// TIA Portal V17 export
// export: Created 2022-07-20T07:01:31.3759363Z, ExportSetting WithDefaults, DisplayName Totally Integrated Automation Portal, DisplayVersion V17, DisplayName TIA Portal Openness, DisplayVersion V17, DisplayName TIA Portal Version Control Interface, DisplayVersion V17, DisplayName SINAMICS Startdrive Advanced, DisplayVersion V17, DisplayName SINAMICS Startdrive G130, G150, S120, S150, SINAMICS MV, S210, DisplayVersion V17, DisplayName SINAMICS Startdrive G110M, G120, G120C, G120D, G120P, G115D, DisplayVersion V17, DisplayName STEP 7 Professional, DisplayVersion V17, DisplayName STEP 7 Safety, DisplayVersion V17, DisplayName WinCC Advanced, DisplayVersion V17
FUNCTION "FC10330_2BytesToUDint" : UDInt   // FC10330, LAD
{ S7_Optimized_Access := 'TRUE' }
VERSION : 0.1
// stored: AutoNumber false, IsIECCheckEnabled false, SetENOAutomatically false, UDAEnableTagReadback false
   VAR_INPUT
      LowByte : Byte;
      HighByte : Byte;
   END_VAR
BEGIN

REGION Network 1 (SCL): 2 Bytes To Udint Conversion
   #FC10330_2BytesToUDint := WORD_TO_UDINT(SHL_WORD(IN := #HighByte, N := 8) OR #LowByte);
END_REGION
END_FUNCTION
